TYPE ST_MTI_STATUS :
STRUCT
  EventCount            : USINT;
  InputState            : BIT;
  InputBufferOverflow   : BIT;
  InputCycleCounter     : ST_2BIT;
  CountsInBuffer        : USINT;
  InputOrderFeedback    : usint;
END_STRUCT
END_TYPE

(* stored: Version 1.1.0.1
   DUT ST_MTI_STATUS: Id {ea99a0e6-9189-4da5-9d3b-fde812558013} *)
